// TIA Portal V16 export
// export: Created 2023-08-28T09:37:29.9515651Z, ExportSetting WithDefaults, DisplayName Totally Integrated Automation Portal, DisplayVersion V16 Update 6, DisplayName TIA Portal Version Control Interface, DisplayVersion V16 Update 2, DisplayName TIA Portal Openness, DisplayVersion V16 Update 6, DisplayName STEP 7 Professional, DisplayVersion V16 Update 6, DisplayName STEP 7 Safety, DisplayVersion V16, DisplayName WinCC Advanced, DisplayVersion V16 Update 6
ORGANIZATION_BLOCK "Cyclic interrupt_2"   // OB32, LAD, CyclicInterrupt
TITLE = Pobranie analogów z wejścia
{ S7_Optimized_Access := 'TRUE' }
AUTHOR : rtecmer
VERSION : 0.1
// Obsługa wejść analogowych
// stored: AutoNumber true, IsIECCheckEnabled false, SetENOAutomatically false
   VAR_INPUT
      Initial_Call : Bool;   // Initial call of this OB
      Event_Count : Int;   // Events discarded
   END_VAR
BEGIN

REGION Network 1: Pobranie wartości z wejść analogowych
   // B6 - Miasto
   // B7 - Pompownia
   // B8 - Suchobieg
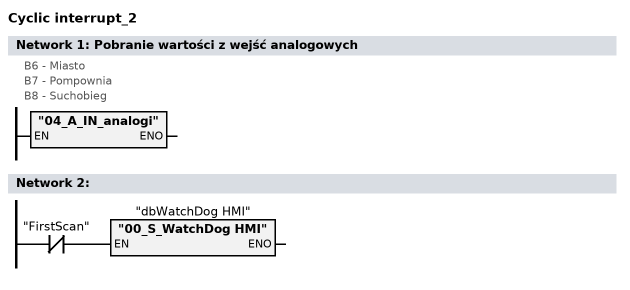
   RUNG wire#powerrail
      "04_A_IN_analogi"()
   END_RUNG
   // the same network as SCL:
   "04_A_IN_analogi"();
END_REGION

REGION Network 2
   RUNG wire#powerrail
      I_Contact( "FirstScan" )
      "dbWatchDog HMI"()
   END_RUNG
   // the same network as SCL:
   IF NOT "FirstScan" THEN
       "dbWatchDog HMI"();   // "00_S_WatchDog HMI"
   END_IF;
END_REGION

REGION Network 3 (SCL): Reset znaczników zbocza wysyłania danych przez TCP
   "memRisingTriger_Data_1" := FALSE;
   "memTrig_Client_Receiving_1" := FALSE;
   "memRisingTriger_Data_2" := FALSE;
   "memTrig_Client_Receiving_2" := FALSE;
   "memRisingTriger_Data_3" := FALSE;
   "memTrig_Client_Receiving_3" := FALSE;
   "memRisingTriger_Data_4" := FALSE;
   "memTrig_Client_Receiving_4" := FALSE;
   "memRisingTriger_Data_5" := FALSE;
   "memTrig_Client_Receiving_5" := FALSE;
   "memRisingTriger_Data_6" := FALSE;
   "memTrig_Client_Receiving_6" := FALSE;
   "memRisingTriger_Data_7" := FALSE;
   "memTrig_Client_Receiving_7" := FALSE;
   "memRisingTriger_Data_8" := FALSE;
   "memTrig_Client_Receiving_8" := FALSE;
   "memRisingTriger_Data_9" := FALSE;
   "memTrig_Client_Receiving_9" := FALSE;
   "memRisingTriger_Data_10" := FALSE;
   "memTrig_Client_Receiving_10" := FALSE;
END_REGION

REGION Network 4 (SCL): pamieć zbocza narastającego przekazania danej do wysłania
   "memRisingTriger_Data_11" := FALSE;
   "memTrig_Client_Receiving_11" := FALSE;
   "memRisingTriger_Data_12" := FALSE;
   "memTrig_Client_Receiving_12" := FALSE;
   "memRisingTriger_Data_13" := FALSE;
   "memTrig_Client_Receiving_13" := FALSE;
   "memRisingTriger_Data_14" := FALSE;
   "memTrig_Client_Receiving_14" := FALSE;
   "memRisingTriger_Data_15" := FALSE;
   "memTrig_Client_Receiving_15" := FALSE;
   "memRisingTriger_Data_16" := FALSE;
   "memTrig_Client_Receiving_16" := FALSE;
   "memRisingTriger_Data_17" := FALSE;
   "memTrig_Client_Receiving_17" := FALSE;
   "memRisingTriger_Data_18" := FALSE;
   "memTrig_Client_Receiving_18" := FALSE;
   "memRisingTriger_Data_19" := FALSE;
   "memTrig_Client_Receiving_19" := FALSE;
   "memRisingTriger_Data_20" := FALSE;
   "memTrig_Client_Receiving_20" := FALSE;
END_REGION
END_ORGANIZATION_BLOCK
